(* IEC 61131-3 sources: learning-path/05_oop_in_st/exercises/3_calculator_current_volume/src, 2 files *)

(* ---- ItfTank.st ---- *)
//File to create the interface to implement the class tank
NAMESPACE FluidHandlingClass

    INTERFACE ItfTank
        METHOD Fill
        END_METHOD
        METHOD Flush
        END_METHOD
        METHOD  Close
        END_METHOD
        METHOD Emptying
        END_METHOD
    END_INTERFACE

END_NAMESPACE

(* ---- basicTank.st ---- *)
NAMESPACE FluidHandlingClass
    class BasicTank IMPLEMENTS ITank
        VAR PUBLIC
            inletValve: ValveClass;
            outletValve: ValveClass;
        END_VAR

        METHOD PRIVATE OpenInlet
            inletValve.Open();
        END_METHOD
        METHOD PRIVATE OpenOutlet
            outletValve.Open();
        END_METHOD
        METHOD PRIVATE CloseInlet
            inletValve.Close();
        END_METHOD
        METHOD PRIVATE CloseOutlet
            outletValve.Close();
        END_METHOD

        METHOD PUBLIC Fill
            this.OpenInlet();
            this.CloseOutlet();
        END_METHOD

        METHOD PUBLIC Flush
            this.OpenInlet();
            this.OpenOutlet();
        END_METHOD

        METHOD PUBLIC Close
            this.CloseInlet();
            this.CloseOutlet();
        END_METHOD

        METHOD PUBLIC Emptying
            this.CloseInlet();
            this.OpenOutlet();
        END_METHOD
    END_CLASS
END_NAMESPACE
